Omron CX-Programmer project NewProject (CX-Programmer 9.61)

# PLC PLC1: CJ2M CPU12

## Global symbols (name address type ; comment)
0.00 BOOL  ; Start
0.01 BOOL  ; Start
0.02 BOOL  ; Start
0.03 BOOL  ; Start
0.04 BOOL  ; Start
0.05 BOOL  ; Start
0.06 BOOL  ; Start
0.07 BOOL  ; Start
0.08 BOOL  ; Start
0.09 BOOL  ; Start
0.10 BOOL  ; Start
0.11 BOOL  ; Start
0.12 BOOL  ; Start
0.13 BOOL  ; Start
0.14 BOOL  ; Start
0.15 BOOL  ; Start
100.00 BOOL  ; Light Panel  G.1
100.01 BOOL  ; Light Panel G.2
100.02 BOOL  ; Light Panel G.3
100.03 BOOL  ; Light Panel G.4
100.04 BOOL  ; Light Panel G.5
100.05 BOOL  ; Light Panel G.6
100.06 BOOL  ; Light Panel G.7
100.07 BOOL  ; Light Panel G.8
100.08 BOOL  ; Light Panel G.9
100.09 BOOL  ; Light Panel G.10
100.10 BOOL  ; Light Panel G.1
100.11 BOOL  ; Light Panel G.2
100.12 BOOL  ; Light Panel G.3
100.13 BOOL  ; Light Panel G.4
100.14 BOOL  ; Light Panel G.5
100.15 BOOL  ; Light Panel G.6
101.00 BOOL  ; Light Panel G.7
101.01 BOOL  ; Light Panel G.8
101.02 BOOL  ; Light Panel G.9
101.03 BOOL  ; Light Panel G.10
101.04 BOOL  ; Light Panel G.11
101.05 BOOL  ; Light Panel G.12
101.06 BOOL  ; Light Panel G.13
101.07 BOOL  ; Light Panel G.14
101.08 BOOL  ; Light Panel G.1
101.09 BOOL  ; Light Panel G.2
101.10 BOOL  ; Light Panel G.3
101.11 BOOL  ; Light Panel G.4
101.12 BOOL  ; Light Panel G.5
101.13 BOOL  ; Light Panel G.6
101.14 BOOL  ; Light Panel G.7
101.15 BOOL  ; Light Panel G.8
102.00 BOOL  ; Light Panel G.9
102.01 BOOL  ; Light Panel G.10
102.02 BOOL  ; Light Panel G.11
102.03 BOOL  ; Light Panel G.12
102.04 BOOL  ; Light Panel G.13
102.05 BOOL  ; Light Panel G.14
102.06 BOOL  ; Light Panel G.15
102.07 BOOL  ; Light Panel G.16
102.08 BOOL  ; Light Panel G.17
102.09 BOOL  ; Light Panel G.18
102.10 BOOL  ; Light Panel G.19
102.11 BOOL  ; Light Panel G.20
102.12 BOOL  ; Light Panel G.1
102.13 BOOL  ; Light Panel G.2
102.14 BOOL  ; Light Panel G.3
102.15 BOOL  ; Light Panel G.4
103.00 BOOL  ; Light Panel G.5
103.01 BOOL  ; Light Panel G.6
103.02 BOOL  ; Light Panel G.7
103.03 BOOL  ; Light Panel G.8
103.04 BOOL  ; Light Panel G.9
103.05 BOOL  ; Light Panel G.10
103.06 BOOL  ; Light Panel G.11
103.07 BOOL  ; Light Panel G.12
103.08 BOOL  ; Light Panel G.13
103.09 BOOL  ; Light Panel G.14
103.10 BOOL  ; Light Panel G.15
103.11 BOOL  ; Light Panel G.16
103.12 BOOL  ; Light Panel G.17
103.13 BOOL  ; Light Panel G.18
103.14 BOOL  ; Light Panel G.19
103.15 BOOL  ; Light Panel G.20
104.00 BOOL  ; Light Panel G.1
104.01 BOOL  ; Light Panel G.2
104.02 BOOL  ; Light Panel G.3
104.03 BOOL  ; Light Panel G.4
104.04 BOOL  ; Light Panel G.5
104.05 BOOL  ; Light Panel G.6
104.06 BOOL  ; Light Panel G.7
104.07 BOOL  ; Light Panel G.8
104.08 BOOL  ; Light Panel G.9
104.09 BOOL  ; Light Panel G.10
104.10 BOOL  ; Light Panel G.11
104.11 BOOL  ; Light Panel G.12
104.12 BOOL  ; Light Panel G.13
104.13 BOOL  ; Light Panel G.14
104.14 BOOL  ; Light Panel G.15
104.15 BOOL  ; Light Panel G.16
105.00 BOOL  ; Light Panel G.17
105.01 BOOL  ; Light Panel G.18
105.02 BOOL  ; Light Panel G.19
105.03 BOOL  ; Light Panel G.20
105.04 BOOL  ; Light Panel G.21
105.05 BOOL  ; Light Panel G.1
105.06 BOOL  ; Light Panel G.2
105.07 BOOL  ; Light Panel G.3
105.08 BOOL  ; Light Panel G.4
105.09 BOOL  ; Light Panel G.5
105.10 BOOL  ; Light Panel G.6
105.11 BOOL  ; Light Panel G.7
105.12 BOOL  ; Light Panel G.8
105.13 BOOL  ; Light Panel G.9
105.14 BOOL  ; Light Panel G.10
105.15 BOOL  ; Light Panel G.11
106.00 BOOL  ; Light Panel G.12
106.01 BOOL  ; Light Panel G.13
106.02 BOOL  ; Light Panel G.14
106.03 BOOL  ; Light Panel G.15
106.04 BOOL  ; Light Panel G.16
106.05 BOOL  ; Light Panel G.17
106.06 BOOL  ; Light Panel G.18
106.07 BOOL  ; Light Panel G.19
106.08 BOOL  ; Light Panel G.20
106.09 BOOL  ; Light Panel G.21
106.10 BOOL  ; Light Panel G.22
106.11 BOOL  ; Light Panel G.23
106.12 BOOL  ; Light Panel G.24
106.13 BOOL  ; Light Panel G.25
106.14 BOOL  ; Light Panel G.26
106.15 BOOL  ; Light Panel G.1
107.00 BOOL  ; Light Panel G.2
107.01 BOOL  ; Light Panel G.3
107.02 BOOL  ; Light Panel G.4
107.03 BOOL  ; Light Panel G.5
107.04 BOOL  ; Light Panel G.6
107.05 BOOL  ; Light Panel G.7
107.06 BOOL  ; Light Panel G.8
107.07 BOOL  ; Light Panel G.9
107.08 BOOL  ; Light Panel G.10
107.09 BOOL  ; Light Panel G.11
107.10 BOOL  ; Light Panel G.12
107.11 BOOL  ; Light Panel G.13
107.12 BOOL  ; Light Panel G.14
107.13 BOOL  ; Light Panel G.15
107.14 BOOL  ; Light Panel G.16
107.15 BOOL  ; Light Panel G.17
108.00 BOOL  ; Light Panel G.18
108.01 BOOL  ; Light Panel G.19
108.02 BOOL  ; Light Panel G.20
108.03 BOOL  ; Light Panel G.21
108.04 BOOL  ; Light Panel G.22
108.05 BOOL  ; Light Panel G.23
108.06 BOOL  ; Light Panel G.1
108.07 BOOL  ; Light Panel G.2
108.08 BOOL  ; Light Panel G.3
108.09 BOOL  ; Light Panel G.4
108.10 BOOL  ; Light Panel G.5
108.11 BOOL  ; Light Panel G.6
108.12 BOOL  ; Light Panel G.7
108.13 BOOL  ; Light Panel G.8
108.14 BOOL  ; Light Panel G.9
108.15 BOOL  ; Light Panel G.10
109.00 BOOL  ; Light Panel G.11
109.01 BOOL  ; Light Panel G.12
109.02 BOOL  ; Light Panel G.13
109.03 BOOL  ; Light Panel G.14
109.04 BOOL  ; Light Panel G.15
109.05 BOOL  ; Light Panel G.16
109.06 BOOL  ; Light Panel G.17
109.07 BOOL  ; Light Panel G.18
109.08 BOOL  ; Light Panel G.19
109.09 BOOL  ; Light Panel G.16
109.10 BOOL  ; Power Panel G.1
109.11 BOOL  ; Power Panel G.2
109.12 BOOL  ; Power Panel G.3
109.13 BOOL  ; Power Panel G.4
109.14 BOOL  ; Power Panel G.5
109.15 BOOL  ; Power Panel G.6
10.00 BOOL  ; Start
10.01 BOOL  ; Start
10.02 BOOL  ; Start
10.03 BOOL  ; Start
10.04 BOOL  ; Start
10.05 BOOL  ; Start
10.06 BOOL  ; Start
10.07 BOOL  ; Start
10.08 BOOL  ; Start
10.09 BOOL  ; Start
10.10 BOOL  ; Start
10.11 BOOL  ; Start
10.12 BOOL  ; Start
10.13 BOOL  ; Start
10.14 BOOL  ; Start
10.15 BOOL  ; Start
110.00 BOOL  ; Power Panel G.7
110.01 BOOL  ; Power Panel G.8
110.02 BOOL  ; Power Panel G.9
110.03 BOOL  ; Power Panel G.10
110.04 BOOL  ; Power Panel G.11
110.05 BOOL  ; Power Panel G.12
110.06 BOOL  ; Light Panel G.1
110.07 BOOL  ; Light Panel G.2
110.08 BOOL  ; Light Panel G.3
110.09 BOOL  ; Light Panel G.4
110.10 BOOL  ; Light Panel G.5
110.11 BOOL  ; Light Panel G.6
110.12 BOOL  ; Light Panel G.7
110.13 BOOL  ; Light Panel G.8
110.14 BOOL  ; Light Panel G.9
110.15 BOOL  ; Light Panel G.10
111.00 BOOL  ; Light Panel G.11
111.01 BOOL  ; Light Panel G.12
111.02 BOOL  ; Light Panel G.13
111.03 BOOL  ; Light Panel G.14
111.04 BOOL  ; Power Panel G.1
111.05 BOOL  ; Power Panel G.2
111.06 BOOL  ; Power Panel G.3
111.07 BOOL  ; Power Panel G.4
111.08 BOOL  ; Power Panel G.5
111.09 BOOL  ; Power Panel G.6
111.10 BOOL  ; Power Panel G.7
111.11 BOOL  ; Power Panel G.8
111.12 BOOL  ; Power Panel G.9
111.13 BOOL  ; Power Panel G.10
111.14 BOOL  ; Power Panel G.11
111.15 BOOL  ; Power Panel G.12
112.00 BOOL  ; Power Panel G.13
112.01 BOOL  ; Power Panel G.14
112.02 BOOL  ; Power Panel G.15
112.03 BOOL  ; Power Panel G.16
112.04 BOOL  ; Power Panel G.17
112.05 BOOL  ; Power Panel G.18
112.06 BOOL  ; Power Panel G.19
112.07 BOOL  ; Power Panel G.20
112.08 BOOL  ; Power Panel G.21
112.09 BOOL  ; Power Panel G.22
112.10 BOOL  ; Power Panel G.23
112.11 BOOL  ; Light Panel G.1
112.12 BOOL  ; Light Panel G.2
112.13 BOOL  ; Light Panel G.3
112.14 BOOL  ; Light Panel G.4
112.15 BOOL  ; Light Panel G.5
113.00 BOOL  ; Light Panel G.6
113.01 BOOL  ; Light Panel G.7
113.02 BOOL  ; Light Panel G.8
113.03 BOOL  ; Light Panel G.9
113.04 BOOL  ; Light Panel G.10
113.05 BOOL  ; Light Panel G.11
113.06 BOOL  ; Light Panel G.12
113.07 BOOL  ; Light Panel G.13
113.08 BOOL  ; Light Panel G.14
113.09 BOOL  ; Light Panel G.15
113.10 BOOL  ; Light Panel G.16
113.11 BOOL  ; Power Panel G.1
113.12 BOOL  ; Power Panel G.2
113.13 BOOL  ; Power Panel G.3
113.14 BOOL  ; Power Panel G.4
113.15 BOOL  ; Power Panel G.5
114.00 BOOL  ; Power Panel G.6
114.01 BOOL  ; Power Panel G.7
114.02 BOOL  ; Power Panel G.8
114.03 BOOL  ; Power Panel G.9
114.04 BOOL  ; Power Panel G.10
114.05 BOOL  ; Power Panel G.11
114.06 BOOL  ; Power Panel G.12
114.07 BOOL  ; Power Panel G.13
114.08 BOOL  ; Power Panel G.14
114.09 BOOL  ; Power Panel G.15
114.10 BOOL  ; Power Panel G.16
114.11 BOOL  ; Power Panel G.17
114.12 BOOL  ; Power Panel G.18
114.13 BOOL  ; Power Panel G.19
114.14 BOOL  ; Power Panel G.20
114.15 BOOL  ; Power Panel G.21
115.00 BOOL  ; Power Panel G.22
115.01 BOOL  ; Power Panel G.22
116.10 BOOL  ; MCB
11.00 BOOL  ; Start
11.01 BOOL  ; Start
11.02 BOOL  ; Start
11.03 BOOL  ; Start
11.04 BOOL  ; Start
11.05 BOOL  ; Start
11.06 BOOL  ; Start
11.07 BOOL  ; Start
11.08 BOOL  ; Start
11.09 BOOL  ; Start
11.10 BOOL  ; Start
11.11 BOOL  ; Start
11.12 BOOL  ; Start
11.13 BOOL  ; Start
11.14 BOOL  ; Start
11.15 BOOL  ; Start
12.00 BOOL  ; Start
12.01 BOOL  ; Start
12.02 BOOL  ; Start
12.03 BOOL  ; Start
12.04 BOOL  ; Start
12.05 BOOL  ; Start
12.06 BOOL  ; Start
12.07 BOOL  ; Start
12.08 BOOL  ; Start
12.09 BOOL  ; Start
12.10 BOOL  ; Start
12.11 BOOL  ; Start
12.12 BOOL  ; Start
12.13 BOOL  ; Start
12.14 BOOL  ; Start
12.15 BOOL  ; Start
13.00 BOOL  ; Start
13.01 BOOL  ; Start
13.02 BOOL  ; Start
13.03 BOOL  ; Start
13.04 BOOL  ; Start
13.05 BOOL  ; Start
13.06 BOOL  ; Start
13.07 BOOL  ; Start
13.08 BOOL  ; Start
13.09 BOOL  ; Start
13.10 BOOL  ; Start
13.11 BOOL  ; Start
13.12 BOOL  ; Start
13.13 BOOL  ; Start
13.14 BOOL  ; Start
13.15 BOOL  ; Start
14.00 BOOL  ; Start
14.01 BOOL  ; Start
14.02 BOOL  ; Start
14.03 BOOL  ; Start
14.04 BOOL  ; Start
14.05 BOOL  ; Start
14.06 BOOL  ; Start
14.07 BOOL  ; Stop
14.08 BOOL  ; Start
14.09 BOOL  ; Stop
14.10 BOOL  ; Start
14.11 BOOL  ; Stop
14.12 BOOL  ; Start
14.13 BOOL  ; Stop
14.14 BOOL  ; Start
14.15 BOOL  ; Stop
15.00 BOOL  ; Start
15.01 BOOL  ; Stop
15.02 BOOL  ; Start
15.03 BOOL  ; Stop
15.04 BOOL  ; Start
15.05 BOOL  ; Stop
15.06 BOOL  ; Start
15.07 BOOL  ; Start
15.08 BOOL  ; Start
15.09 BOOL  ; Start
15.10 BOOL  ; Start
15.11 BOOL  ; Start
15.12 BOOL  ; Start
15.13 BOOL  ; Start
15.14 BOOL  ; Start
15.15 BOOL  ; Start
16.00 BOOL  ; Start
16.01 BOOL  ; Stop
16.02 BOOL  ; Start
16.03 BOOL  ; Stop
16.04 BOOL  ; Start
16.05 BOOL  ; Stop
16.06 BOOL  ; Start
16.07 BOOL  ; Stop
16.08 BOOL  ; Start
16.09 BOOL  ; Stop
16.10 BOOL  ; Start
16.11 BOOL  ; Stop
16.12 BOOL  ; Start
16.13 BOOL  ; Stop
16.14 BOOL  ; Start
16.15 BOOL  ; Stop
17.00 BOOL  ; Start
17.01 BOOL  ; Stop
17.02 BOOL  ; Start
17.03 BOOL  ; Stop
17.04 BOOL  ; Start
17.05 BOOL  ; Stop
17.06 BOOL  ; Start
17.07 BOOL  ; Stop
17.08 BOOL  ; Start
17.09 BOOL  ; Stop
17.10 BOOL  ; Start
17.11 BOOL  ; Stop
17.12 BOOL  ; Start
17.13 BOOL  ; Stop
17.14 BOOL  ; Start
17.15 BOOL  ; Stop
18.00 BOOL  ; Start
18.01 BOOL  ; Stop
18.02 BOOL  ; Start
18.03 BOOL  ; Stop
18.04 BOOL  ; Start
18.05 BOOL  ; Stop
18.06 BOOL  ; Start
18.07 BOOL  ; Stop
18.08 BOOL  ; Start
18.09 BOOL  ; Stop
18.10 BOOL  ; Start
18.11 BOOL  ; Stop
18.12 BOOL  ; Start
18.13 BOOL  ; Stop
18.14 BOOL  ; Start
18.15 BOOL  ; Stop
19.00 BOOL  ; Start
19.01 BOOL  ; Stop
19.02 BOOL  ; Start
19.03 BOOL  ; Stop
19.04 BOOL  ; Start
19.05 BOOL  ; Stop
19.06 BOOL  ; Start
19.07 BOOL  ; Stop
19.08 BOOL  ; Start
19.09 BOOL  ; Stop
19.10 BOOL  ; Start
19.11 BOOL  ; Stop
19.12 BOOL  ; Start
19.13 BOOL  ; Stop
19.14 BOOL  ; Start
19.15 BOOL  ; Stop
1.00 BOOL  ; Start
1.01 BOOL  ; Start
1.02 BOOL  ; Start
1.03 BOOL  ; Start
1.04 BOOL  ; Start
1.05 BOOL  ; Start
1.06 BOOL  ; Start
1.07 BOOL  ; Start
1.08 BOOL  ; Start
1.09 BOOL  ; Start
1.10 BOOL  ; Start
1.11 BOOL  ; Start
1.12 BOOL  ; Start
1.13 BOOL  ; Start
1.14 BOOL  ; Start
1.15 BOOL  ; Start
208.14 BOOL  ; Light Panel G.9
20.00 BOOL  ; Start
20.01 BOOL  ; Stop
20.02 BOOL  ; Start
20.03 BOOL  ; Stop
20.04 BOOL  ; Start
20.05 BOOL  ; Stop
20.06 BOOL  ; Start
20.07 BOOL  ; Stop
20.08 BOOL  ; Start
20.09 BOOL  ; Stop
20.10 BOOL  ; Start
20.11 BOOL  ; Stop
20.12 BOOL  ; Start
20.13 BOOL  ; Stop
20.14 BOOL  ; Start
20.15 BOOL  ; Stop
21.00 BOOL  ; Start
21.01 BOOL  ; Stop
21.02 BOOL  ; Start
21.03 BOOL  ; Stop
21.04 BOOL  ; Start
21.05 BOOL  ; Stop
21.06 BOOL  ; Start
21.07 BOOL  ; Stop
21.08 BOOL  ; Start
21.09 BOOL  ; Stop
21.10 BOOL  ; Start
21.11 BOOL  ; Stop
21.12 BOOL  ; Start
21.13 BOOL  ; Stop
21.14 BOOL  ; Start
21.15 BOOL  ; Stop
22.00 BOOL  ; Start
22.01 BOOL  ; Stop
22.02 BOOL  ; Start
22.03 BOOL  ; Stop
22.04 BOOL  ; Start
22.05 BOOL  ; Stop
22.06 BOOL  ; Start
22.07 BOOL  ; Stop
22.08 BOOL  ; Start
22.09 BOOL  ; Stop
22.10 BOOL  ; Start
22.11 BOOL  ; Stop
22.12 BOOL  ; Start
22.13 BOOL  ; Stop
22.14 BOOL  ; Start
22.15 BOOL  ; Stop
23.00 BOOL  ; Start
23.01 BOOL  ; Stop
23.02 BOOL  ; Start
23.03 BOOL  ; Stop
23.04 BOOL  ; Start
23.05 BOOL  ; Stop
23.06 BOOL  ; Start
23.07 BOOL  ; Stop
23.08 BOOL  ; Start
23.09 BOOL  ; Stop
23.10 BOOL  ; Start
23.11 BOOL  ; Stop
23.12 BOOL  ; Start
23.13 BOOL  ; Stop
23.14 BOOL  ; Start
23.15 BOOL  ; Stop
24.00 BOOL  ; Start
24.01 BOOL  ; Stop
24.02 BOOL  ; Start
24.03 BOOL  ; Stop
24.04 BOOL  ; Start
24.05 BOOL  ; Stop
24.06 BOOL  ; Start
24.07 BOOL  ; Stop
24.08 BOOL  ; Start
24.09 BOOL  ; Stop
24.10 BOOL  ; Start
24.11 BOOL  ; Stop
24.12 BOOL  ; Start
24.13 BOOL  ; Stop
24.14 BOOL  ; Start
24.15 BOOL  ; Stop
25.00 BOOL  ; Start
25.01 BOOL  ; Stop
25.02 BOOL  ; Start
25.03 BOOL  ; Stop
25.04 BOOL  ; Start
25.05 BOOL  ; Stop
25.06 BOOL  ; Start
25.07 BOOL  ; Stop
25.08 BOOL  ; Start
25.09 BOOL  ; Stop
25.10 BOOL  ; Start
25.11 BOOL  ; Stop
25.12 BOOL  ; Start
25.13 BOOL  ; Stop
25.14 BOOL  ; Start
25.15 BOOL  ; Stop
26.00 BOOL  ; Start
26.01 BOOL  ; Stop
26.02 BOOL  ; Start
26.03 BOOL  ; Stop
26.04 BOOL  ; Start
26.05 BOOL  ; Stop
26.06 BOOL  ; Start
26.07 BOOL  ; Stop
26.08 BOOL  ; Start
26.09 BOOL  ; Stop
26.10 BOOL  ; Start
26.11 BOOL  ; Stop
26.12 BOOL  ; Start
26.13 BOOL  ; Stop
26.14 BOOL  ; Start
26.15 BOOL  ; Stop
27.00 BOOL  ; Start
27.01 BOOL  ; Stop
27.02 BOOL  ; Start
27.03 BOOL  ; Stop
27.04 BOOL  ; Start
27.05 BOOL  ; Stop
27.06 BOOL  ; Start
27.07 BOOL  ; Stop
27.08 BOOL  ; Start
27.09 BOOL  ; Stop
27.10 BOOL  ; Start
27.11 BOOL  ; Stop
27.12 BOOL  ; Start
27.13 BOOL  ; Stop
27.14 BOOL  ; Start
27.15 BOOL  ; Stop
28.00 BOOL  ; Start
28.01 BOOL  ; Stop
28.02 BOOL  ; Start
28.03 BOOL  ; Stop
28.04 BOOL  ; Start
28.05 BOOL  ; Stop
28.06 BOOL  ; Start
28.07 BOOL  ; Stop
28.08 BOOL  ; Start
28.09 BOOL  ; Stop
28.10 BOOL  ; Start
28.11 BOOL  ; Stop
28.12 BOOL  ; Start
28.13 BOOL  ; Stop
28.14 BOOL  ; Start
28.15 BOOL  ; Stop
29.00 BOOL  ; Start
29.01 BOOL  ; Stop
29.02 BOOL  ; Start
29.03 BOOL  ; Stop
29.04 BOOL  ; Start
29.05 BOOL  ; Stop
29.06 BOOL  ; Start
29.07 BOOL  ; Stop
29.08 BOOL  ; Start
29.09 BOOL  ; Stop
29.10 BOOL  ; Start
29.11 BOOL  ; Stop
29.12 BOOL  ; Start
29.13 BOOL  ; Stop
29.14 BOOL  ; Start
29.15 BOOL  ; Stop
2.00 BOOL  ; Start
2.01 BOOL  ; Start
2.02 BOOL  ; Start
2.03 BOOL  ; Start
2.04 BOOL  ; Start
2.05 BOOL  ; Start
2.06 BOOL  ; Start
2.07 BOOL  ; Start
2.08 BOOL  ; Start
2.09 BOOL  ; Start
2.10 BOOL  ; Start
2.11 BOOL  ; Start
2.12 BOOL  ; Start
2.13 BOOL  ; Start
2.14 BOOL  ; Start
2.15 BOOL  ; Start
30.00 BOOL  ; Start
30.01 BOOL  ; Stop
30.02 BOOL  ; Tanggal/Jam Off
30.03 BOOL  ; Menit/Detik
30.04 BOOL  ; Tanggal/Jam On
30.05 BOOL  ; Tanggal/Jam Off
30.06 BOOL  ; Menit/Detik
30.07 BOOL  ; Tanggal/Jam On
30.08 BOOL  ; Tanggal/Jam Off
30.09 BOOL  ; Menit/Detik
30.10 BOOL  ; Tanggal/Jam On
30.11 BOOL  ; Tanggal/Jam Off
30.12 BOOL  ; Menit/Detik
30.13 BOOL  ; Tanggal/Jam On
30.14 BOOL  ; Tanggal/Jam Off
30.15 BOOL  ; Menit/Detik
31.00 BOOL  ; Tanggal/Jam On
31.01 BOOL  ; Tanggal/Jam Off
31.02 BOOL  ; Timer
31.03 BOOL  ; Menit/Detik
31.04 BOOL  ; Tanggal/Jam On
31.05 BOOL  ; Tanggal/Jam Off
31.06 BOOL  ; Menit/Detik
31.07 BOOL  ; Tanggal/Jam On
31.08 BOOL  ; Tanggal/Jam Off
31.09 BOOL  ; Menit/Detik
31.10 BOOL  ; Tanggal/Jam On
31.11 BOOL  ; Tanggal/Jam Off
31.12 BOOL  ; Meniit/Detik
31.13 BOOL  ; Tanggal/Jam On
31.14 BOOL  ; Tanggal/Jam Off
31.15 BOOL  ; Menit/Detik
32.00 BOOL  ; Tanggal/Jam On
32.01 BOOL  ; Tanggal/Jam Off
32.02 BOOL  ; Menit/Detik
32.03 BOOL  ; Tanggal/Jam On
32.04 BOOL  ; Tanggal/Jam Off
32.05 BOOL  ; Menit/Detik
32.06 BOOL  ; Tanggal/Jam On
32.07 BOOL  ; Tanggal/Jam Off
32.08 BOOL  ; Timer
32.09 BOOL  ; Menit/Detik
32.10 BOOL  ; Tanggal/Jam On
32.11 BOOL  ; Tanggal/Jam Off
32.12 BOOL  ; Menit/Detik
32.13 BOOL  ; Tanggal/Jam On
32.14 BOOL  ; Tanggal/Jam Off
32.15 BOOL  ; Menit/Detik
33.00 BOOL  ; Tanggal/Jam On
33.01 BOOL  ; Tanggal/Jam Off
33.02 BOOL  ; Meniit/Detik
33.03 BOOL  ; Tanggal/Jam On
33.04 BOOL  ; Tanggal/Jam Off
33.05 BOOL  ; Menit/Detik
33.06 BOOL  ; Tanggal/Jam On
33.07 BOOL  ; Tanggal/Jam Off
33.08 BOOL  ; Menit/Detik
33.09 BOOL  ; Tanggal/Jam On
33.10 BOOL  ; Tanggal/Jam Off
33.11 BOOL  ; Menit/Detik
33.12 BOOL  ; Tanggal/Jam On
33.13 BOOL  ; Tanggal/Jam Off
33.14 BOOL  ; Timer
33.15 BOOL  ; Menit/Detik
34.00 BOOL  ; Tanggal/Jam On
34.01 BOOL  ; Tanggal/Jam Off
34.02 BOOL  ; Menit/Detik
34.03 BOOL  ; Tanggal/Jam On
34.04 BOOL  ; Tanggal/Jam Off
34.05 BOOL  ; Menit/Detik
34.06 BOOL  ; Tanggal/Jam On
34.07 BOOL  ; Tanggal/Jam Off
34.08 BOOL  ; Meniit/Detik
34.09 BOOL  ; Tanggal/Jam On
34.10 BOOL  ; Tanggal/Jam Off
34.11 BOOL  ; Menit/Detik
34.12 BOOL  ; Tanggal/Jam On
34.13 BOOL  ; Tanggal/Jam Off
34.14 BOOL  ; Menit/Detik
34.15 BOOL  ; Tanggal/Jam On
35.00 BOOL  ; Tanggal/Jam Off
35.01 BOOL  ; Menit/Detik
35.02 BOOL  ; Tanggal/Jam On
35.03 BOOL  ; Tanggal/Jam Off
35.04 BOOL  ; Timer
35.05 BOOL  ; Menit/Detik
35.06 BOOL  ; Tanggal/Jam On
35.07 BOOL  ; Tanggal/Jam Off
35.08 BOOL  ; Menit/Detik
35.09 BOOL  ; Tanggal/Jam On
35.10 BOOL  ; Tanggal/Jam Off
35.11 BOOL  ; Menit/Detik
35.12 BOOL  ; Tanggal/Jam On
35.13 BOOL  ; Tanggal/Jam Off
35.14 BOOL  ; Meniit/Detik
35.15 BOOL  ; Tanggal/Jam On
36.00 BOOL  ; Tanggal/Jam Off
36.01 BOOL  ; Menit/Detik
36.02 BOOL  ; Tanggal/Jam On
36.03 BOOL  ; Tanggal/Jam Off
36.04 BOOL  ; Menit/Detik
36.05 BOOL  ; Tanggal/Jam On
36.06 BOOL  ; Tanggal/Jam Off
36.07 BOOL  ; Menit/Detik
36.08 BOOL  ; Tanggal/Jam On
36.09 BOOL  ; Tanggal/Jam Off
3.00 BOOL  ; Start
3.01 BOOL  ; Start
3.02 BOOL  ; Start
3.03 BOOL  ; Start
3.04 BOOL  ; Start
3.05 BOOL  ; Start
3.06 BOOL  ; Start
3.07 BOOL  ; Start
3.08 BOOL  ; Start
3.09 BOOL  ; Start
3.10 BOOL  ; Start
3.11 BOOL  ; Start
3.12 BOOL  ; Start
3.13 BOOL  ; Start
3.14 BOOL  ; Start
3.15 BOOL  ; Start
4.00 BOOL  ; Start
4.01 BOOL  ; Start
4.02 BOOL  ; Start
4.03 BOOL  ; Start
4.04 BOOL  ; Start
4.05 BOOL  ; Start
4.06 BOOL  ; Start
4.07 BOOL  ; Start
4.08 BOOL  ; Start
4.09 BOOL  ; Start
4.10 BOOL  ; Start
4.11 BOOL  ; Start
4.12 BOOL  ; Start
4.13 BOOL  ; Start
4.14 BOOL  ; Start
4.15 BOOL  ; Start
50.00 BOOL  ; MCCB
50.01 BOOL  ; MCCB
50.02 BOOL  ; MCCB
50.03 BOOL  ; MCCB
50.04 BOOL  ; MCCB
50.05 BOOL  ; MCCB
50.06 BOOL  ; MCCB
50.07 BOOL  ; MCCB
50.08 BOOL  ; MCCB
50.09 BOOL  ; MCCB
50.10 BOOL  ; MCB
50.11 BOOL  ; MCB
50.12 BOOL  ; MCB
50.13 BOOL  ; MCB
50.14 BOOL  ; MCCB
50.15 BOOL  ; MCCB
51.00 BOOL  ; MCCB
51.01 BOOL  ; MCCB
51.02 BOOL  ; MCCB
51.03 BOOL  ; MCCB
51.04 BOOL  ; MCCB
51.05 BOOL  ; MCCB
51.06 BOOL  ; MCCB
51.07 BOOL  ; MCCB
51.08 BOOL  ; MCCB
51.09 BOOL  ; MCCB
51.10 BOOL  ; MCCB
51.11 BOOL  ; MCCB
51.12 BOOL  ; MCB
51.13 BOOL  ; MCB
51.14 BOOL  ; MCB
51.15 BOOL  ; MCB
52.00 BOOL  ; MCB
52.01 BOOL  ; MCB
52.02 BOOL  ; MCB
52.03 BOOL  ; MCB
52.04 BOOL  ; MCB
52.05 BOOL  ; MCB
52.06 BOOL  ; MCB
52.07 BOOL  ; MCB
52.08 BOOL  ; MCB
52.09 BOOL  ; MCB
52.10 BOOL  ; MCB
52.11 BOOL  ; MCB
52.12 BOOL  ; MCB
52.13 BOOL  ; MCB
52.14 BOOL  ; MCB
52.15 BOOL  ; MCB
53.00 BOOL  ; MCB
53.01 BOOL  ; MCB
53.02 BOOL  ; MCB
53.03 BOOL  ; MCB
53.04 BOOL  ; MCB
53.05 BOOL  ; MCB
53.06 BOOL  ; MCB
53.07 BOOL  ; MCB
53.08 BOOL  ; MCB
53.09 BOOL  ; MCB
53.10 BOOL  ; MCB
53.11 BOOL  ; MCB
53.12 BOOL  ; MCB
53.13 BOOL  ; MCB
53.14 BOOL  ; MCB
53.15 BOOL  ; MCB
54.00 BOOL  ; MCB
54.01 BOOL  ; MCB
54.02 BOOL  ; MCB
54.03 BOOL  ; MCB
54.04 BOOL  ; MCB
54.05 BOOL  ; MCB
54.06 BOOL  ; MCB
54.07 BOOL  ; MCB
54.08 BOOL  ; MCB
54.09 BOOL  ; MCB
54.10 BOOL  ; MCB
54.11 BOOL  ; MCB
54.12 BOOL  ; MCB
54.13 BOOL  ; MCB
54.14 BOOL  ; MCB
54.15 BOOL  ; MCB
55.00 BOOL  ; MCB
55.01 BOOL  ; MCB
55.02 BOOL  ; MCB
55.03 BOOL  ; MCB
55.04 BOOL  ; MCB
55.05 BOOL  ; MCB
55.06 BOOL  ; MCB
55.07 BOOL  ; MCB
55.08 BOOL  ; MCB
55.09 BOOL  ; MCB
55.10 BOOL  ; MCB
55.11 BOOL  ; MCB
55.12 BOOL  ; MCB
55.13 BOOL  ; MCB
55.14 BOOL  ; MCB
55.15 BOOL  ; MCB
56.00 BOOL  ; MCB
56.01 BOOL  ; MCB
56.02 BOOL  ; MCB
56.03 BOOL  ; MCB
56.04 BOOL  ; MCB
56.05 BOOL  ; MCB
56.06 BOOL  ; MCB
56.07 BOOL  ; MCB
56.08 BOOL  ; MCB
56.09 BOOL  ; MCB
56.10 BOOL  ; MCB
56.11 BOOL  ; MCB
56.12 BOOL  ; MCB
56.13 BOOL  ; MCB
56.14 BOOL  ; MCB
56.15 BOOL  ; MCB
57.00 BOOL  ; MCB
57.01 BOOL  ; MCB
57.02 BOOL  ; MCB
57.03 BOOL  ; MCB
57.04 BOOL  ; MCB
57.05 BOOL  ; MCB
57.06 BOOL  ; MCB
57.07 BOOL  ; MCB
57.08 BOOL  ; MCB
57.09 BOOL  ; MCB
57.10 BOOL  ; MCB
57.11 BOOL  ; MCB
57.12 BOOL  ; MCB
57.13 BOOL  ; MCB
57.14 BOOL  ; MCB
57.15 BOOL  ; MCB
58.00 BOOL  ; MCB
58.01 BOOL  ; MCB
58.02 BOOL  ; MCB
58.03 BOOL  ; MCB
58.04 BOOL  ; MCB
58.05 BOOL  ; MCB
58.06 BOOL  ; MCB
58.07 BOOL  ; MCB
58.08 BOOL  ; MCB
58.09 BOOL  ; MCB
58.10 BOOL  ; MCB
58.11 BOOL  ; MCB
58.12 BOOL  ; MCB
58.13 BOOL  ; MCB
58.14 BOOL  ; MCB
58.15 BOOL  ; MCB
59.00 BOOL  ; MCB
59.01 BOOL  ; MCB
59.02 BOOL  ; MCB
59.03 BOOL  ; MCB
59.04 BOOL  ; MCB
59.05 BOOL  ; MCB
59.06 BOOL  ; MCB
59.07 BOOL  ; MCB
59.08 BOOL  ; MCB
59.09 BOOL  ; MCB
59.10 BOOL  ; MCB
59.11 BOOL  ; MCB
59.12 BOOL  ; MCB
59.13 BOOL  ; MCB
59.14 BOOL  ; MCB
59.15 BOOL  ; MCB
5.00 BOOL  ; Start
5.01 BOOL  ; Start
5.02 BOOL  ; Start
5.03 BOOL  ; Start
5.04 BOOL  ; Start
5.05 BOOL  ; Start
5.06 BOOL  ; Start
5.07 BOOL  ; Start
5.08 BOOL  ; Start
5.09 BOOL  ; Start
5.10 BOOL  ; Start
5.11 BOOL  ; Start
5.12 BOOL  ; Start
5.13 BOOL  ; Start
5.14 BOOL  ; Start
5.15 BOOL  ; Start
60.00 BOOL  ; MCB
60.01 BOOL  ; MCB
60.02 BOOL  ; MCB
60.03 BOOL  ; MCB
60.04 BOOL  ; MCB
60.05 BOOL  ; MCB
60.06 BOOL  ; MCB
60.07 BOOL  ; MCB
60.08 BOOL  ; MCB
60.09 BOOL  ; MCB
60.10 BOOL  ; MCB
60.11 BOOL  ; MCB
60.12 BOOL  ; MCB
60.13 BOOL  ; MCB
60.14 BOOL  ; MCB
60.15 BOOL  ; MCB
61.00 BOOL  ; MCB
61.01 BOOL  ; MCB
61.02 BOOL  ; MCB
61.03 BOOL  ; MCB
61.04 BOOL  ; MCB
61.05 BOOL  ; MCB
61.06 BOOL  ; MCB
61.07 BOOL  ; MCB
61.08 BOOL  ; MCB
61.09 BOOL  ; MCB
61.10 BOOL  ; MCB
61.11 BOOL  ; MCB
61.12 BOOL  ; MCB
61.13 BOOL  ; MCB
61.14 BOOL  ; MCB
61.15 BOOL  ; MCB
62.00 BOOL  ; MCB
62.01 BOOL  ; MCB
62.02 BOOL  ; MCB
62.03 BOOL  ; MCB
62.04 BOOL  ; MCB
62.05 BOOL  ; MCB
62.06 BOOL  ; MCB
62.07 BOOL  ; MCB
62.08 BOOL  ; MCB
62.09 BOOL  ; MCB
62.10 BOOL  ; MCB
62.11 BOOL  ; MCB
62.12 BOOL  ; MCB
62.13 BOOL  ; MCB
62.14 BOOL  ; MCB
62.15 BOOL  ; MCB
63.00 BOOL  ; MCB
63.01 BOOL  ; MCB
63.02 BOOL  ; MCB
63.03 BOOL  ; MCB
63.04 BOOL  ; MCB
63.05 BOOL  ; MCB
63.06 BOOL  ; MCB
63.07 BOOL  ; MCB
63.08 BOOL  ; MCB
63.09 BOOL  ; MCB
63.10 BOOL  ; MCB
63.11 BOOL  ; MCB
63.12 BOOL  ; MCB
63.13 BOOL  ; MCB
63.14 BOOL  ; MCB
63.15 BOOL  ; MCB
64.00 BOOL  ; MCB
64.01 BOOL  ; MCB
64.02 BOOL  ; MCB
64.03 BOOL  ; MCB
64.04 BOOL  ; MCB
64.05 BOOL  ; MCB
64.06 BOOL  ; MCB
64.07 BOOL  ; MCB
64.08 BOOL  ; MCB
64.09 BOOL  ; MCB
64.10 BOOL  ; MCB
64.11 BOOL  ; MCB
64.12 BOOL  ; MCB
64.13 BOOL  ; MCB
64.14 BOOL  ; MCB
64.15 BOOL  ; MCB
65.00 BOOL  ; MCB
6.00 BOOL  ; Start
6.01 BOOL  ; Start
6.02 BOOL  ; Start
6.03 BOOL  ; Start
6.04 BOOL  ; Start
6.05 BOOL  ; Start
6.06 BOOL  ; Start
6.07 BOOL  ; Stop
6.08 BOOL  ; Start
6.09 BOOL  ; Start
6.10 BOOL  ; Start
6.11 BOOL  ; Start
6.12 BOOL  ; Start
6.13 BOOL  ; Start
6.14 BOOL  ; Start
6.15 BOOL  ; Start
70.00 BOOL  ; SDP
70.01 BOOL  ; SDP
70.02 BOOL  ; MCB
70.03 BOOL  ; SDP
70.04 BOOL  ; SDP
70.05 BOOL  ; SDP
70.06 BOOL  ; SDP
70.07 BOOL  ; SDP
70.08 BOOL  ; SDP
70.09 BOOL  ; SDP
70.10 BOOL  ; SDP
70.11 BOOL  ; SDP
70.12 BOOL  ; SDP
70.13 BOOL  ; SDP
70.14 BOOL  ; SDP
70.15 BOOL  ; SDP
7.00 BOOL  ; Start
7.01 BOOL  ; Start
7.02 BOOL  ; Start
7.03 BOOL  ; Start
7.04 BOOL  ; Start
7.05 BOOL  ; Start
7.06 BOOL  ; Start
7.07 BOOL  ; Start
7.08 BOOL  ; Start
7.09 BOOL  ; Start
7.10 BOOL  ; Start
7.11 BOOL  ; Start
7.12 BOOL  ; Start
7.13 BOOL  ; Start
7.14 BOOL  ; Start
7.15 BOOL  ; Start
8.00 BOOL  ; Start
8.01 BOOL  ; Start
8.02 BOOL  ; Start
8.03 BOOL  ; Start
8.04 BOOL  ; Start
8.05 BOOL  ; Start
8.06 BOOL  ; Start
8.07 BOOL  ; Start
8.08 BOOL  ; Start
8.09 BOOL  ; Start
8.10 BOOL  ; Start
8.11 BOOL  ; Start
8.12 BOOL  ; Start
8.13 BOOL  ; Start
8.14 BOOL  ; Start
8.15 BOOL  ; Start
9.00 BOOL  ; Start
9.01 BOOL  ; Start
9.02 BOOL  ; Start
9.03 BOOL  ; Start
9.04 BOOL  ; Start
9.05 BOOL  ; Start
9.06 BOOL  ; Start
9.07 BOOL  ; Start
9.08 BOOL  ; Start
9.09 BOOL  ; Start
9.10 BOOL  ; Start
9.11 BOOL  ; Start
9.12 BOOL  ; Start
9.13 BOOL  ; Start
9.14 BOOL  ; Start
9.15 BOOL  ; Start
T0001 BOOL  ; timer G.1
T0002 BOOL  ; T2
T0003 BOOL  ; timer saklar G.2
T0004 BOOL  ; T4
T0005 BOOL  ; Timer G.3
T0006 BOOL  ; T6
T0007 BOOL  ; Timer G.4
T0008 BOOL  ; T8
T0009 BOOL  ; Timer G.5
T0010 BOOL  ; T10
T0011 BOOL  ; Timer G.6
T0012 BOOL  ; T12
T0013 BOOL  ; Timer G.7
T0014 BOOL  ; T14
T0015 BOOL  ; Timer G.8
T0016 BOOL  ; T16
T0017 BOOL  ; Timer G.9
T0018 BOOL  ; T18
T0019 BOOL  ; Timer G.10
T0020 BOOL  ; T20
T0021 BOOL  ; Timer G.11
T0022 BOOL  ; T22
T0023 BOOL  ; Timer G.12
T0024 BOOL  ; T24
T0025 BOOL  ; Timer G.13
T0026 BOOL  ; T26
T0027 BOOL  ; Timer G.14
T0028 BOOL  ; T28

## Program Kontrol_Lampu (cyclic task 0)
Local symbols
Stop BOOL
q10000 BOOL

### Section Lantai_LG

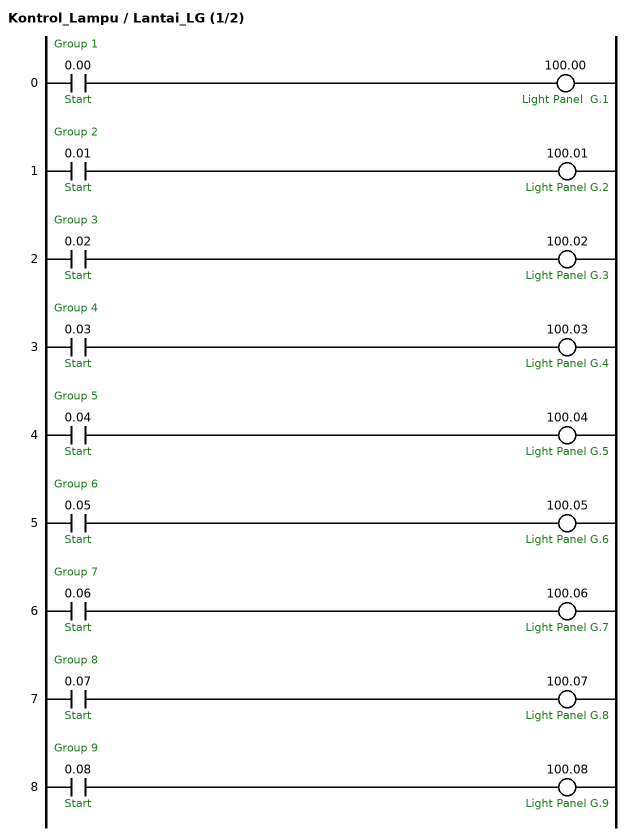
; rung 0: Group 1
LD 0.00  ; Start
OUT 100.00  ; Light Panel  G.1
; rung 1: Group 2
LD 0.01  ; Start
OUT 100.01  ; Light Panel G.2
; rung 2: Group 3
LD 0.02  ; Start
OUT 100.02  ; Light Panel G.3
; rung 3: Group 4
LD 0.03  ; Start
OUT 100.03  ; Light Panel G.4
; rung 4: Group 5
LD 0.04  ; Start
OUT 100.04  ; Light Panel G.5
; rung 5: Group 6
LD 0.05  ; Start
OUT 100.05  ; Light Panel G.6
; rung 6: Group 7
LD 0.06  ; Start
OUT 100.06  ; Light Panel G.7
; rung 7: Group 8
LD 0.07  ; Start
OUT 100.07  ; Light Panel G.8
; rung 8: Group 9
LD 0.08  ; Start
OUT 100.08  ; Light Panel G.9

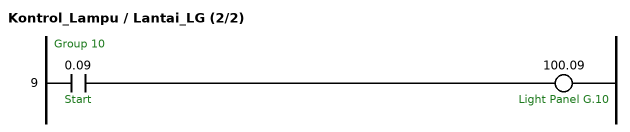
; rung 9: Group 10
LD 0.09  ; Start
OUT 100.09  ; Light Panel G.10

### Section Lantai_1

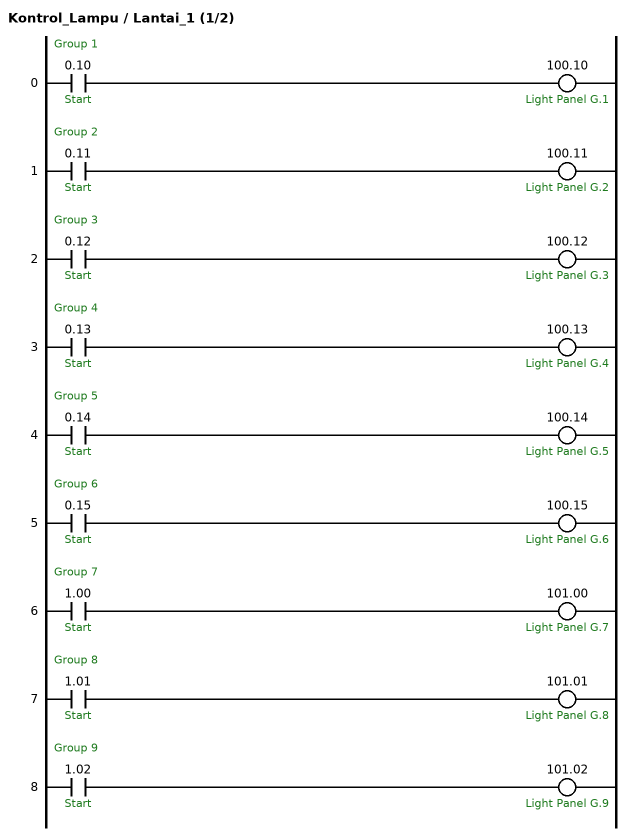
; rung 0: Group 1
LD 0.10  ; Start
OUT 100.10  ; Light Panel G.1
; rung 1: Group 2
LD 0.11  ; Start
OUT 100.11  ; Light Panel G.2
; rung 2: Group 3
LD 0.12  ; Start
OUT 100.12  ; Light Panel G.3
; rung 3: Group 4
LD 0.13  ; Start
OUT 100.13  ; Light Panel G.4
; rung 4: Group 5
LD 0.14  ; Start
OUT 100.14  ; Light Panel G.5
; rung 5: Group 6
LD 0.15  ; Start
OUT 100.15  ; Light Panel G.6
; rung 6: Group 7
LD 1.00  ; Start
OUT 101.00  ; Light Panel G.7
; rung 7: Group 8
LD 1.01  ; Start
OUT 101.01  ; Light Panel G.8
; rung 8: Group 9
LD 1.02  ; Start
OUT 101.02  ; Light Panel G.9

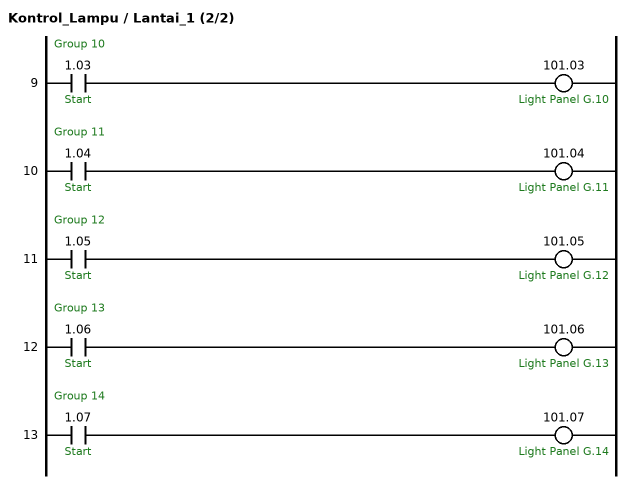
; rung 9: Group 10
LD 1.03  ; Start
OUT 101.03  ; Light Panel G.10
; rung 10: Group 11
LD 1.04  ; Start
OUT 101.04  ; Light Panel G.11
; rung 11: Group 12
LD 1.05  ; Start
OUT 101.05  ; Light Panel G.12
; rung 12: Group 13
LD 1.06  ; Start
OUT 101.06  ; Light Panel G.13
; rung 13: Group 14
LD 1.07  ; Start
OUT 101.07  ; Light Panel G.14

### Section Lantai_2

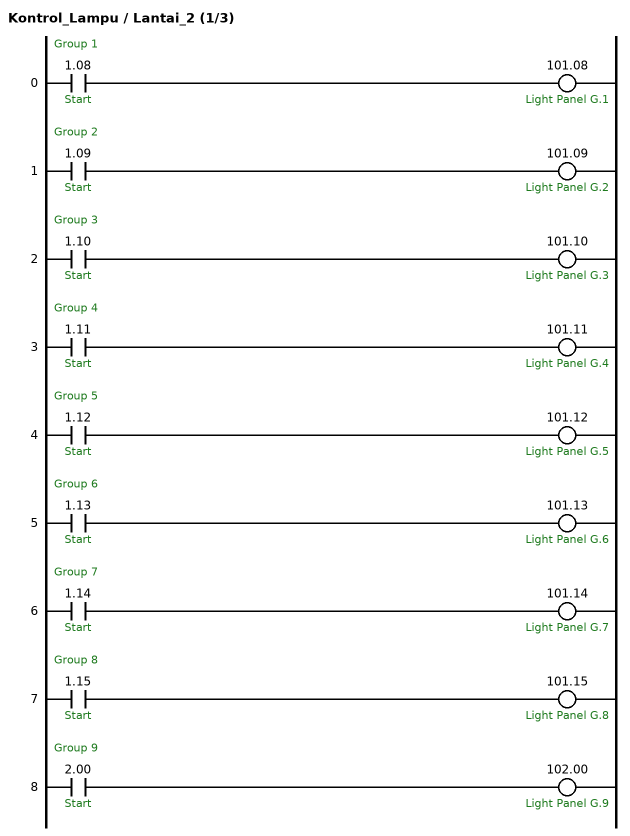
; rung 0: Group 1
LD 1.08  ; Start
OUT 101.08  ; Light Panel G.1
; rung 1: Group 2
LD 1.09  ; Start
OUT 101.09  ; Light Panel G.2
; rung 2: Group 3
LD 1.10  ; Start
OUT 101.10  ; Light Panel G.3
; rung 3: Group 4
LD 1.11  ; Start
OUT 101.11  ; Light Panel G.4
; rung 4: Group 5
LD 1.12  ; Start
OUT 101.12  ; Light Panel G.5
; rung 5: Group 6
LD 1.13  ; Start
OUT 101.13  ; Light Panel G.6
; rung 6: Group 7
LD 1.14  ; Start
OUT 101.14  ; Light Panel G.7
; rung 7: Group 8
LD 1.15  ; Start
OUT 101.15  ; Light Panel G.8
; rung 8: Group 9
LD 2.00  ; Start
OUT 102.00  ; Light Panel G.9

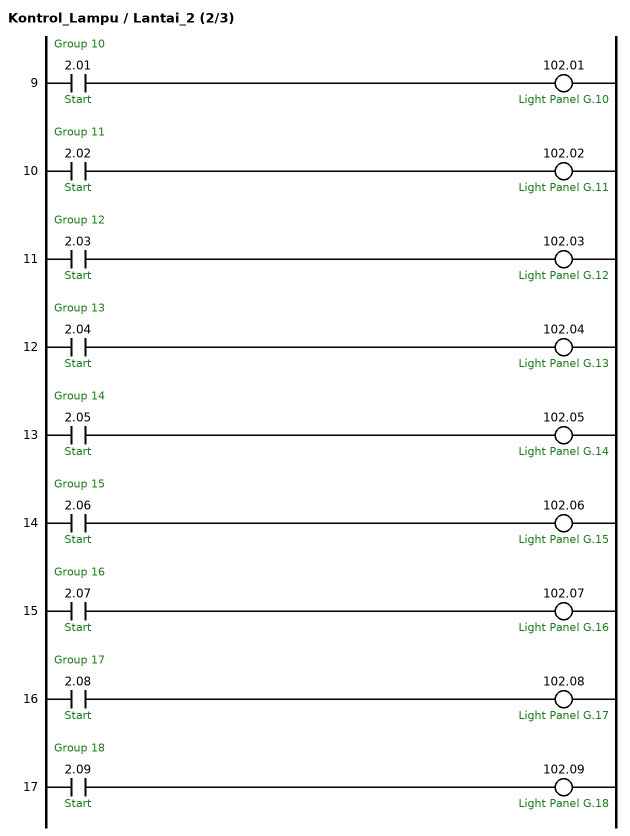
; rung 9: Group 10
LD 2.01  ; Start
OUT 102.01  ; Light Panel G.10
; rung 10: Group 11
LD 2.02  ; Start
OUT 102.02  ; Light Panel G.11
; rung 11: Group 12
LD 2.03  ; Start
OUT 102.03  ; Light Panel G.12
; rung 12: Group 13
LD 2.04  ; Start
OUT 102.04  ; Light Panel G.13
; rung 13: Group 14
LD 2.05  ; Start
OUT 102.05  ; Light Panel G.14
; rung 14: Group 15
LD 2.06  ; Start
OUT 102.06  ; Light Panel G.15
; rung 15: Group 16
LD 2.07  ; Start
OUT 102.07  ; Light Panel G.16
; rung 16: Group 17
LD 2.08  ; Start
OUT 102.08  ; Light Panel G.17
; rung 17: Group 18
LD 2.09  ; Start
OUT 102.09  ; Light Panel G.18

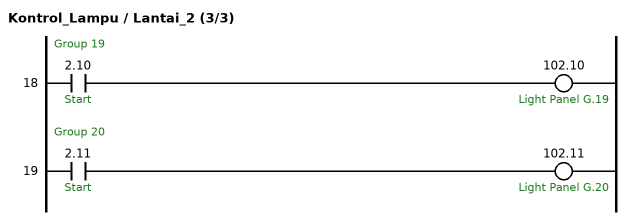
; rung 18: Group 19
LD 2.10  ; Start
OUT 102.10  ; Light Panel G.19
; rung 19: Group 20
LD 2.11  ; Start
OUT 102.11  ; Light Panel G.20

### Section Lantai_3

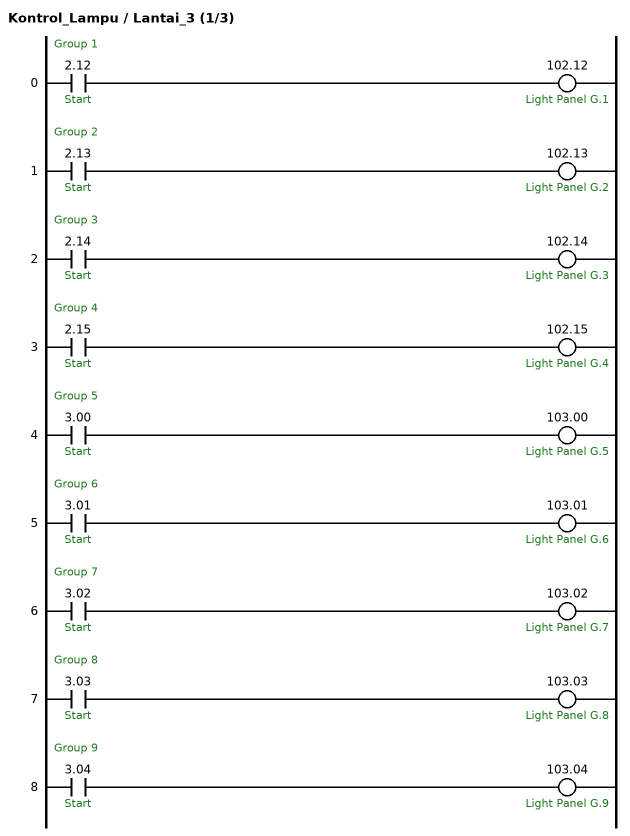
; rung 0: Group 1
LD 2.12  ; Start
OUT 102.12  ; Light Panel G.1
; rung 1: Group 2
LD 2.13  ; Start
OUT 102.13  ; Light Panel G.2
; rung 2: Group 3
LD 2.14  ; Start
OUT 102.14  ; Light Panel G.3
; rung 3: Group 4
LD 2.15  ; Start
OUT 102.15  ; Light Panel G.4
; rung 4: Group 5
LD 3.00  ; Start
OUT 103.00  ; Light Panel G.5
; rung 5: Group 6
LD 3.01  ; Start
OUT 103.01  ; Light Panel G.6
; rung 6: Group 7
LD 3.02  ; Start
OUT 103.02  ; Light Panel G.7
; rung 7: Group 8
LD 3.03  ; Start
OUT 103.03  ; Light Panel G.8
; rung 8: Group 9
LD 3.04  ; Start
OUT 103.04  ; Light Panel G.9

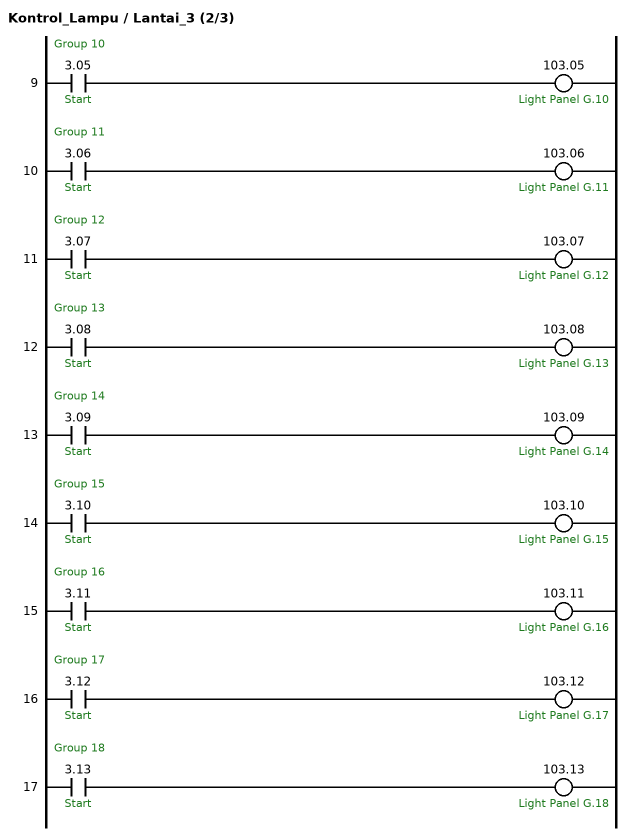
; rung 9: Group 10
LD 3.05  ; Start
OUT 103.05  ; Light Panel G.10
; rung 10: Group 11
LD 3.06  ; Start
OUT 103.06  ; Light Panel G.11
; rung 11: Group 12
LD 3.07  ; Start
OUT 103.07  ; Light Panel G.12
; rung 12: Group 13
LD 3.08  ; Start
OUT 103.08  ; Light Panel G.13
; rung 13: Group 14
LD 3.09  ; Start
OUT 103.09  ; Light Panel G.14
; rung 14: Group 15
LD 3.10  ; Start
OUT 103.10  ; Light Panel G.15
; rung 15: Group 16
LD 3.11  ; Start
OUT 103.11  ; Light Panel G.16
; rung 16: Group 17
LD 3.12  ; Start
OUT 103.12  ; Light Panel G.17
; rung 17: Group 18
LD 3.13  ; Start
OUT 103.13  ; Light Panel G.18

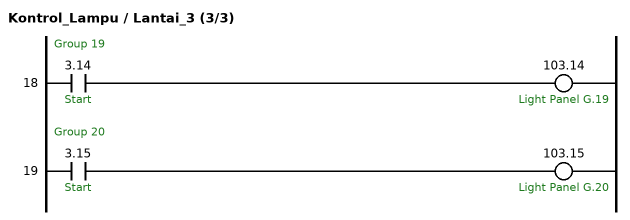
; rung 18: Group 19
LD 3.14  ; Start
OUT 103.14  ; Light Panel G.19
; rung 19: Group 20
LD 3.15  ; Start
OUT 103.15  ; Light Panel G.20

### Section Lantai_4

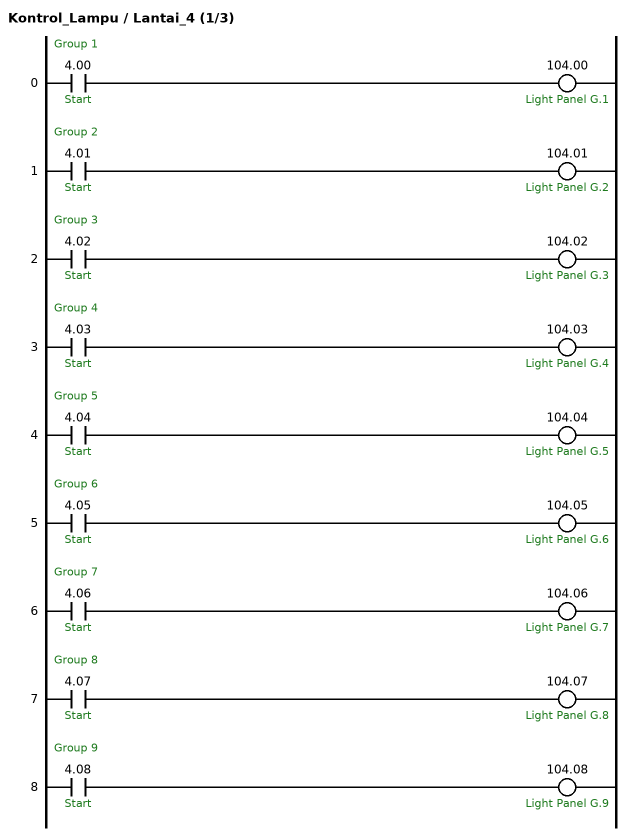
; rung 0: Group 1
LD 4.00  ; Start
OUT 104.00  ; Light Panel G.1
; rung 1: Group 2
LD 4.01  ; Start
OUT 104.01  ; Light Panel G.2
; rung 2: Group 3
LD 4.02  ; Start
OUT 104.02  ; Light Panel G.3
; rung 3: Group 4
LD 4.03  ; Start
OUT 104.03  ; Light Panel G.4
; rung 4: Group 5
LD 4.04  ; Start
OUT 104.04  ; Light Panel G.5
; rung 5: Group 6
LD 4.05  ; Start
OUT 104.05  ; Light Panel G.6
; rung 6: Group 7
LD 4.06  ; Start
OUT 104.06  ; Light Panel G.7
; rung 7: Group 8
LD 4.07  ; Start
OUT 104.07  ; Light Panel G.8
; rung 8: Group 9
LD 4.08  ; Start
OUT 104.08  ; Light Panel G.9

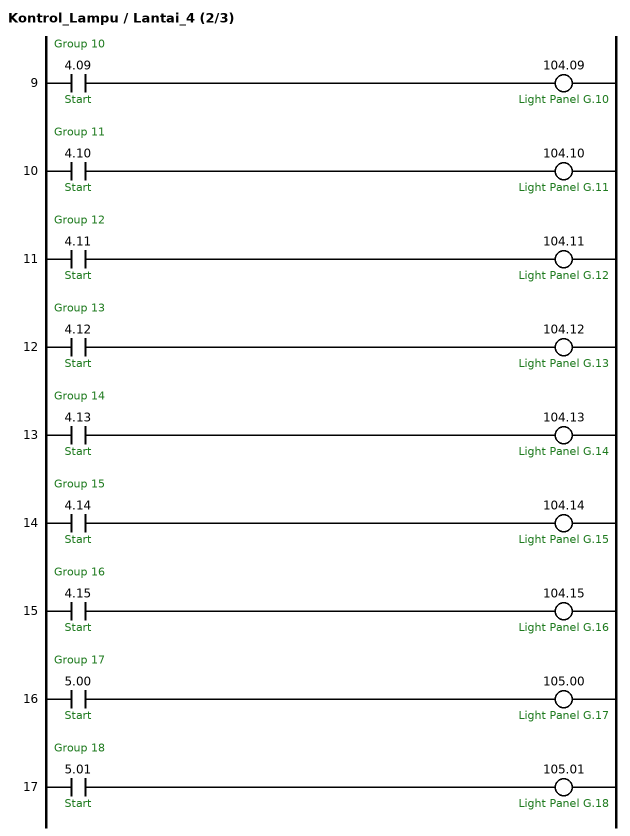
; rung 9: Group 10
LD 4.09  ; Start
OUT 104.09  ; Light Panel G.10
; rung 10: Group 11
LD 4.10  ; Start
OUT 104.10  ; Light Panel G.11
; rung 11: Group 12
LD 4.11  ; Start
OUT 104.11  ; Light Panel G.12
; rung 12: Group 13
LD 4.12  ; Start
OUT 104.12  ; Light Panel G.13
; rung 13: Group 14
LD 4.13  ; Start
OUT 104.13  ; Light Panel G.14
; rung 14: Group 15
LD 4.14  ; Start
OUT 104.14  ; Light Panel G.15
; rung 15: Group 16
LD 4.15  ; Start
OUT 104.15  ; Light Panel G.16
; rung 16: Group 17
LD 5.00  ; Start
OUT 105.00  ; Light Panel G.17
; rung 17: Group 18
LD 5.01  ; Start
OUT 105.01  ; Light Panel G.18

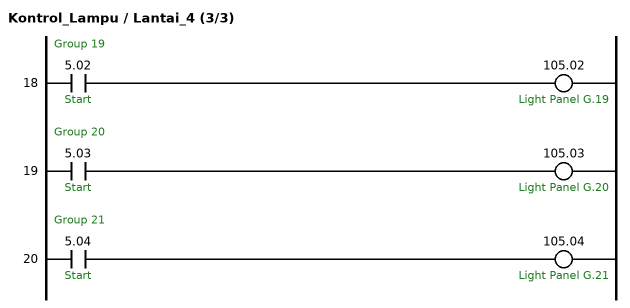
; rung 18: Group 19
LD 5.02  ; Start
OUT 105.02  ; Light Panel G.19
; rung 19: Group 20
LD 5.03  ; Start
OUT 105.03  ; Light Panel G.20
; rung 20: Group 21
LD 5.04  ; Start
OUT 105.04  ; Light Panel G.21

### Section Lantai_5

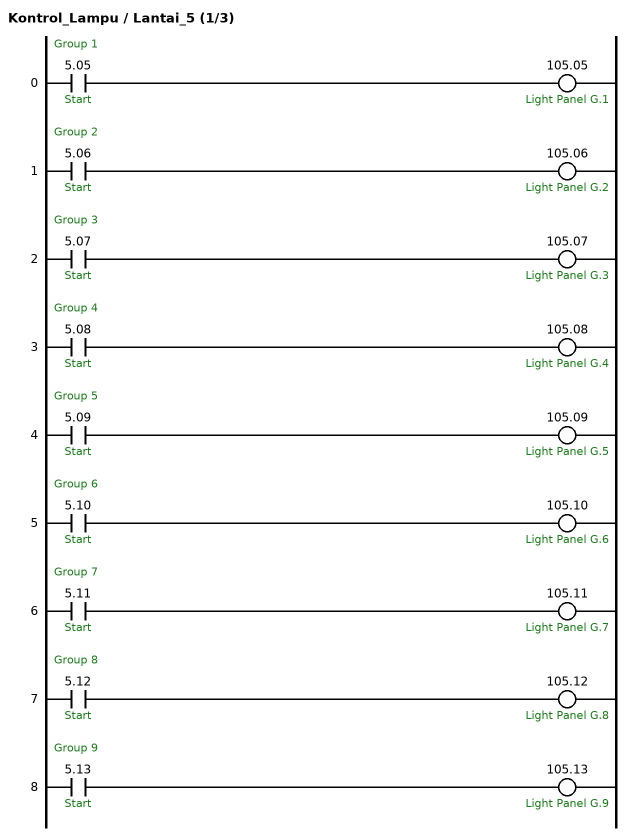
; rung 0: Group 1
LD 5.05  ; Start
OUT 105.05  ; Light Panel G.1
; rung 1: Group 2
LD 5.06  ; Start
OUT 105.06  ; Light Panel G.2
; rung 2: Group 3
LD 5.07  ; Start
OUT 105.07  ; Light Panel G.3
; rung 3: Group 4
LD 5.08  ; Start
OUT 105.08  ; Light Panel G.4
; rung 4: Group 5
LD 5.09  ; Start
OUT 105.09  ; Light Panel G.5
; rung 5: Group 6
LD 5.10  ; Start
OUT 105.10  ; Light Panel G.6
; rung 6: Group 7
LD 5.11  ; Start
OUT 105.11  ; Light Panel G.7
; rung 7: Group 8
LD 5.12  ; Start
OUT 105.12  ; Light Panel G.8
; rung 8: Group 9
LD 5.13  ; Start
OUT 105.13  ; Light Panel G.9

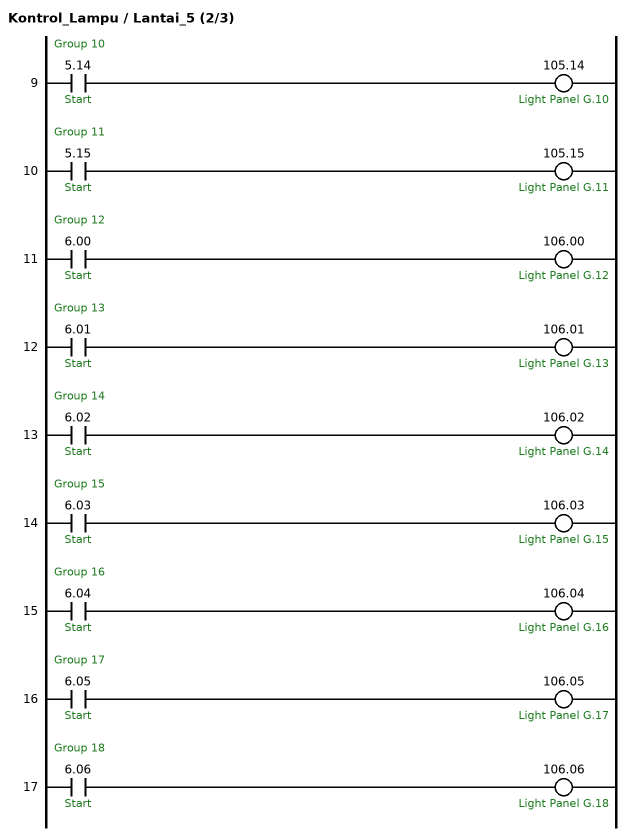
; rung 9: Group 10
LD 5.14  ; Start
OUT 105.14  ; Light Panel G.10
; rung 10: Group 11
LD 5.15  ; Start
OUT 105.15  ; Light Panel G.11
; rung 11: Group 12
LD 6.00  ; Start
OUT 106.00  ; Light Panel G.12
; rung 12: Group 13
LD 6.01  ; Start
OUT 106.01  ; Light Panel G.13
; rung 13: Group 14
LD 6.02  ; Start
OUT 106.02  ; Light Panel G.14
; rung 14: Group 15
LD 6.03  ; Start
OUT 106.03  ; Light Panel G.15
; rung 15: Group 16
LD 6.04  ; Start
OUT 106.04  ; Light Panel G.16
; rung 16: Group 17
LD 6.05  ; Start
OUT 106.05  ; Light Panel G.17
; rung 17: Group 18
LD 6.06  ; Start
OUT 106.06  ; Light Panel G.18

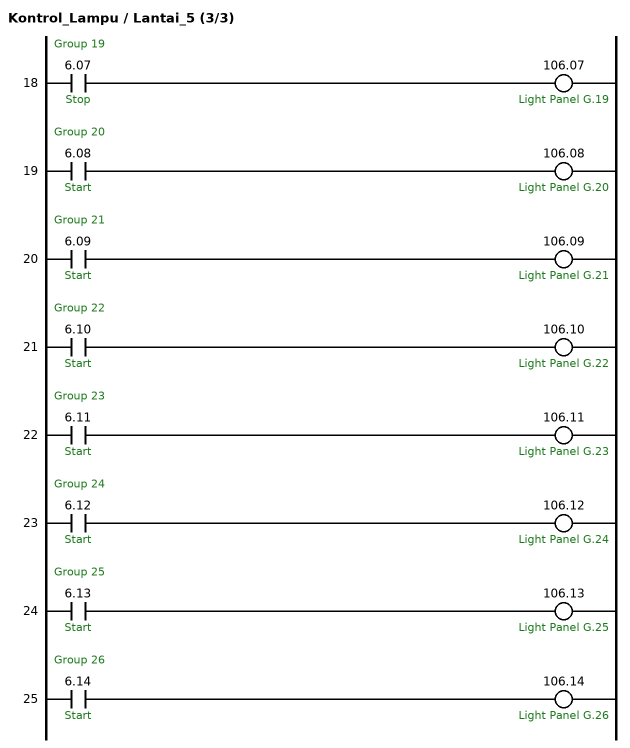
; rung 18: Group 19
LD 6.07  ; Stop
OUT 106.07  ; Light Panel G.19
; rung 19: Group 20
LD 6.08  ; Start
OUT 106.08  ; Light Panel G.20
; rung 20: Group 21
LD 6.09  ; Start
OUT 106.09  ; Light Panel G.21
; rung 21: Group 22
LD 6.10  ; Start
OUT 106.10  ; Light Panel G.22
; rung 22: Group 23
LD 6.11  ; Start
OUT 106.11  ; Light Panel G.23
; rung 23: Group 24
LD 6.12  ; Start
OUT 106.12  ; Light Panel G.24
; rung 24: Group 25
LD 6.13  ; Start
OUT 106.13  ; Light Panel G.25
; rung 25: Group 26
LD 6.14  ; Start
OUT 106.14  ; Light Panel G.26

### Section Lantai_6

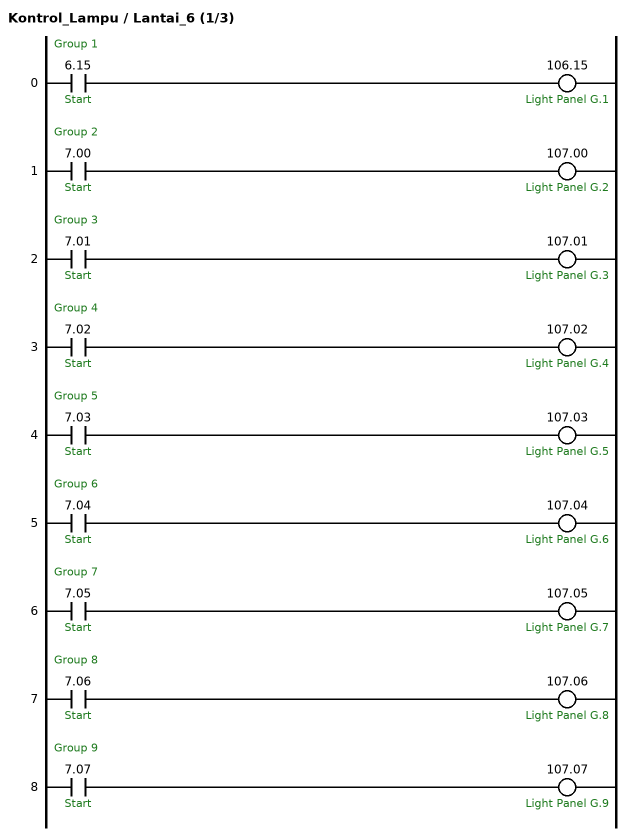
; rung 0: Group 1
LD 6.15  ; Start
OUT 106.15  ; Light Panel G.1
; rung 1: Group 2
LD 7.00  ; Start
OUT 107.00  ; Light Panel G.2
; rung 2: Group 3
LD 7.01  ; Start
OUT 107.01  ; Light Panel G.3
; rung 3: Group 4
LD 7.02  ; Start
OUT 107.02  ; Light Panel G.4
; rung 4: Group 5
LD 7.03  ; Start
OUT 107.03  ; Light Panel G.5
; rung 5: Group 6
LD 7.04  ; Start
OUT 107.04  ; Light Panel G.6
; rung 6: Group 7
LD 7.05  ; Start
OUT 107.05  ; Light Panel G.7
; rung 7: Group 8
LD 7.06  ; Start
OUT 107.06  ; Light Panel G.8
; rung 8: Group 9
LD 7.07  ; Start
OUT 107.07  ; Light Panel G.9

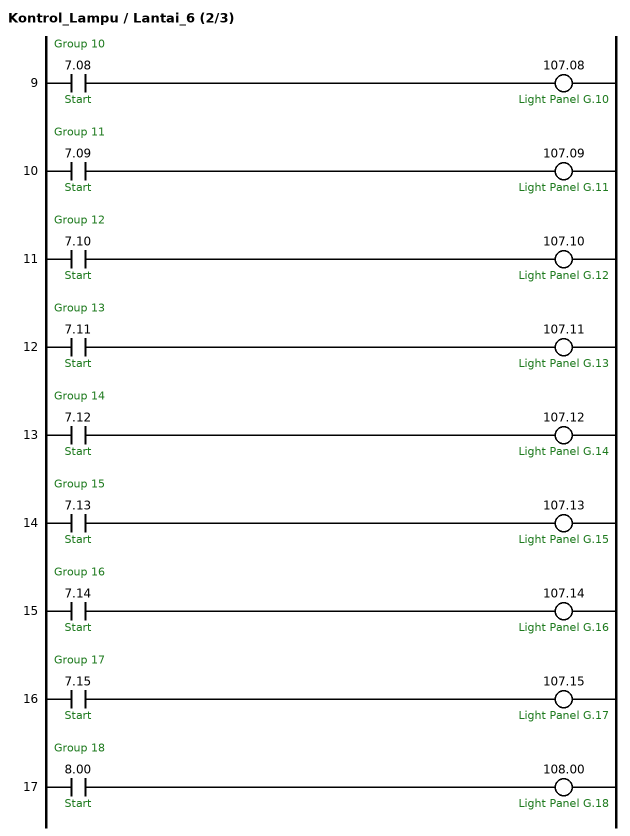
; rung 9: Group 10
LD 7.08  ; Start
OUT 107.08  ; Light Panel G.10
; rung 10: Group 11
LD 7.09  ; Start
OUT 107.09  ; Light Panel G.11
; rung 11: Group 12
LD 7.10  ; Start
OUT 107.10  ; Light Panel G.12
; rung 12: Group 13
LD 7.11  ; Start
OUT 107.11  ; Light Panel G.13
; rung 13: Group 14
LD 7.12  ; Start
OUT 107.12  ; Light Panel G.14
; rung 14: Group 15
LD 7.13  ; Start
OUT 107.13  ; Light Panel G.15
; rung 15: Group 16
LD 7.14  ; Start
OUT 107.14  ; Light Panel G.16
; rung 16: Group 17
LD 7.15  ; Start
OUT 107.15  ; Light Panel G.17
; rung 17: Group 18
LD 8.00  ; Start
OUT 108.00  ; Light Panel G.18

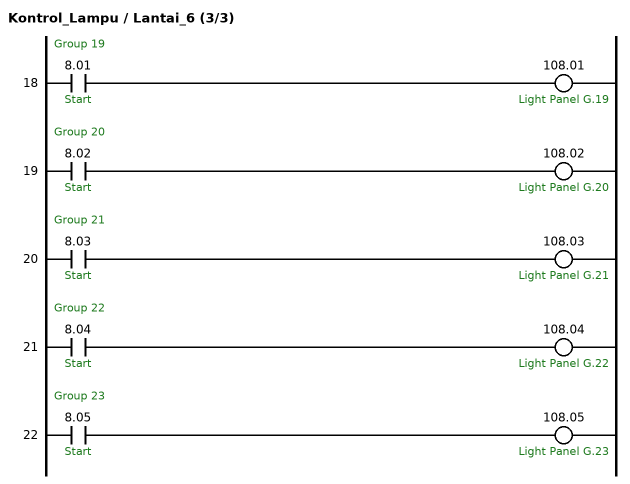
; rung 18: Group 19
LD 8.01  ; Start
OUT 108.01  ; Light Panel G.19
; rung 19: Group 20
LD 8.02  ; Start
OUT 108.02  ; Light Panel G.20
; rung 20: Group 21
LD 8.03  ; Start
OUT 108.03  ; Light Panel G.21
; rung 21: Group 22
LD 8.04  ; Start
OUT 108.04  ; Light Panel G.22
; rung 22: Group 23
LD 8.05  ; Start
OUT 108.05  ; Light Panel G.23

### Section Lantai_7

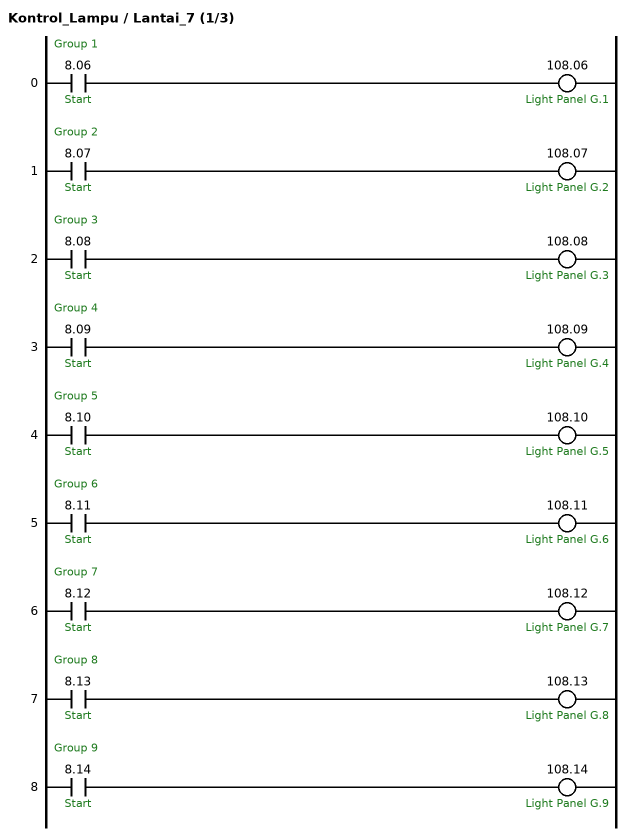
; rung 0: Group 1
LD 8.06  ; Start
OUT 108.06  ; Light Panel G.1
; rung 1: Group 2
LD 8.07  ; Start
OUT 108.07  ; Light Panel G.2
; rung 2: Group 3
LD 8.08  ; Start
OUT 108.08  ; Light Panel G.3
; rung 3: Group 4
LD 8.09  ; Start
OUT 108.09  ; Light Panel G.4
; rung 4: Group 5
LD 8.10  ; Start
OUT 108.10  ; Light Panel G.5
; rung 5: Group 6
LD 8.11  ; Start
OUT 108.11  ; Light Panel G.6
; rung 6: Group 7
LD 8.12  ; Start
OUT 108.12  ; Light Panel G.7
; rung 7: Group 8
LD 8.13  ; Start
OUT 108.13  ; Light Panel G.8
; rung 8: Group 9
LD 8.14  ; Start
OUT 108.14  ; Light Panel G.9

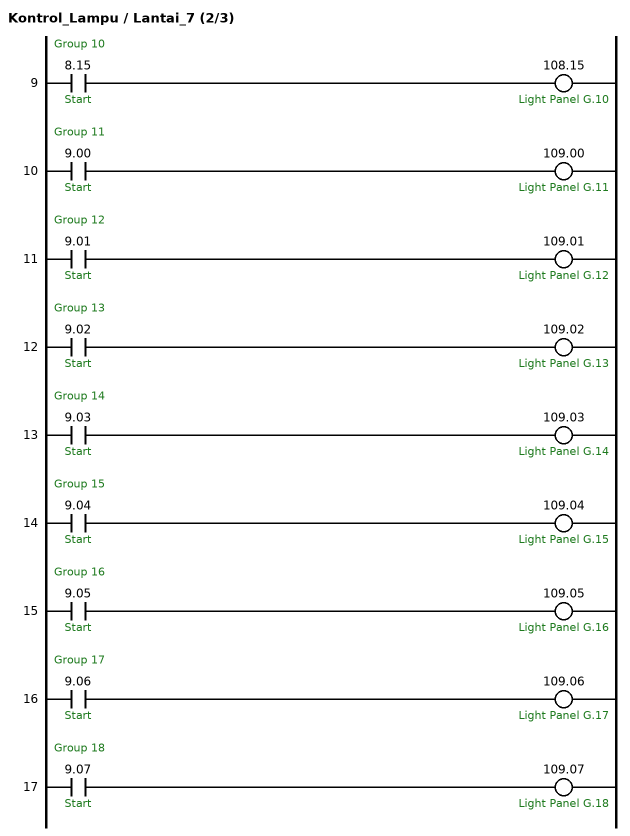
; rung 9: Group 10
LD 8.15  ; Start
OUT 108.15  ; Light Panel G.10
; rung 10: Group 11
LD 9.00  ; Start
OUT 109.00  ; Light Panel G.11
; rung 11: Group 12
LD 9.01  ; Start
OUT 109.01  ; Light Panel G.12
; rung 12: Group 13
LD 9.02  ; Start
OUT 109.02  ; Light Panel G.13
; rung 13: Group 14
LD 9.03  ; Start
OUT 109.03  ; Light Panel G.14
; rung 14: Group 15
LD 9.04  ; Start
OUT 109.04  ; Light Panel G.15
; rung 15: Group 16
LD 9.05  ; Start
OUT 109.05  ; Light Panel G.16
; rung 16: Group 17
LD 9.06  ; Start
OUT 109.06  ; Light Panel G.17
; rung 17: Group 18
LD 9.07  ; Start
OUT 109.07  ; Light Panel G.18

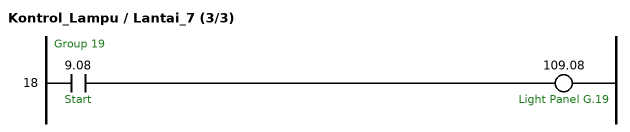
; rung 18: Group 19
LD 9.08  ; Start
OUT 109.08  ; Light Panel G.19

### Section Phasa_R

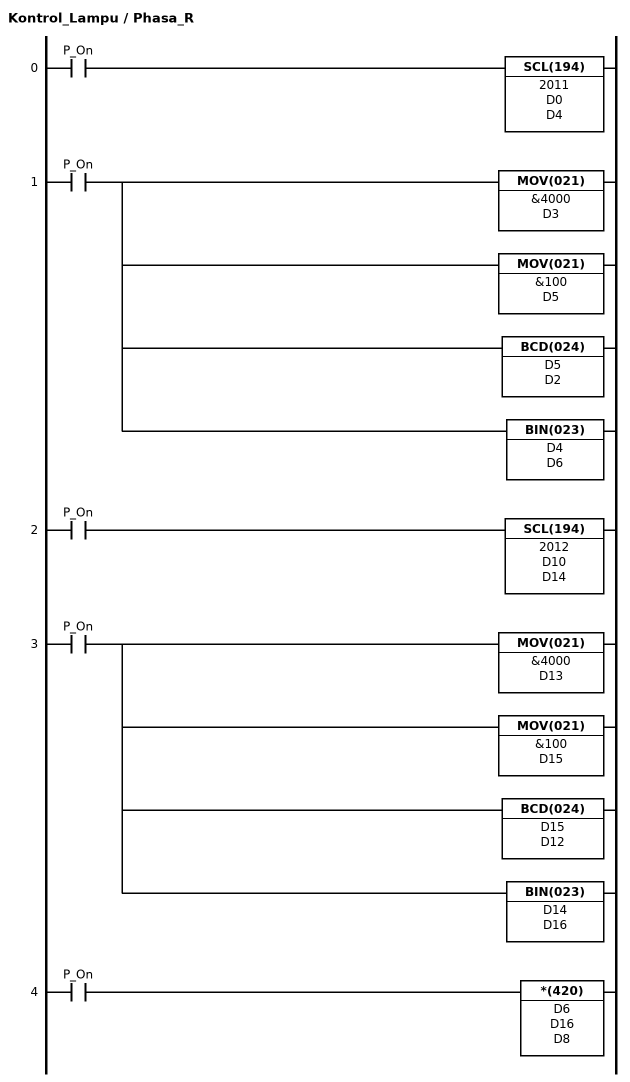
; rung 0
LD P_On
SCL(194) 2011 D0 D4
; rung 1
LD P_On
MOV(021) &4000 D3
MOV(021) &100 D5
BCD(024) D5 D2
BIN(023) D4 D6
; rung 2
LD P_On
SCL(194) 2012 D10 D14
; rung 3
LD P_On
MOV(021) &4000 D13
MOV(021) &100 D15
BCD(024) D15 D12
BIN(023) D14 D16
; rung 4
LD P_On
*(420) D6 D16 D8

### Section Phasa_S

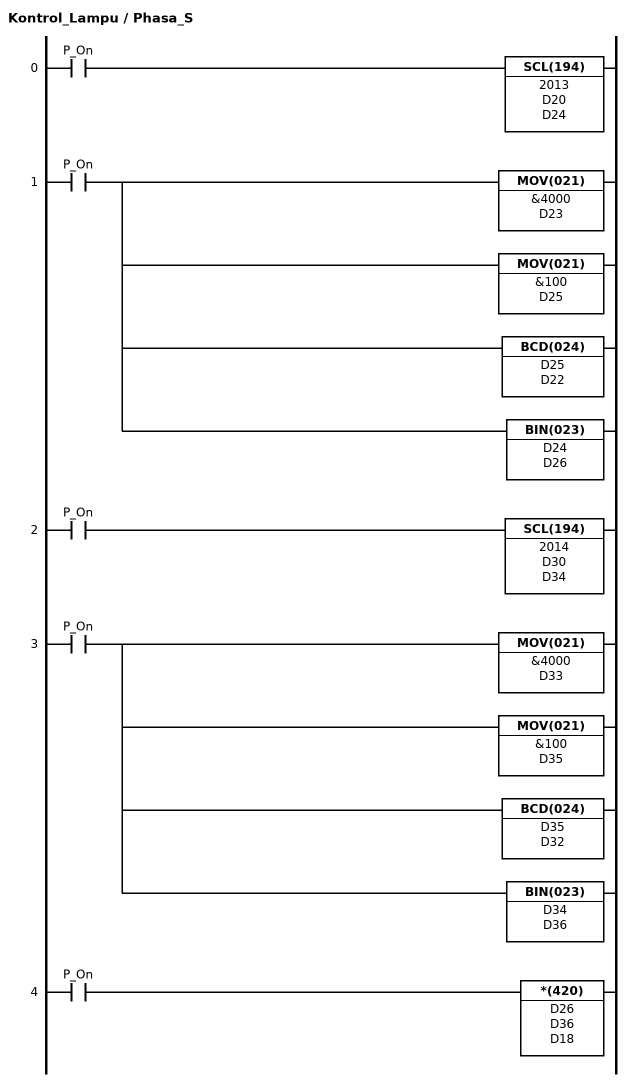
; rung 0
LD P_On
SCL(194) 2013 D20 D24
; rung 1
LD P_On
MOV(021) &4000 D23
MOV(021) &100 D25
BCD(024) D25 D22
BIN(023) D24 D26
; rung 2
LD P_On
SCL(194) 2014 D30 D34
; rung 3
LD P_On
MOV(021) &4000 D33
MOV(021) &100 D35
BCD(024) D35 D32
BIN(023) D34 D36
; rung 4
LD P_On
*(420) D26 D36 D18

### Section Phasa_T

